TYPE E_CircuitBreakerStatus :
(
    READY := 0,         // Hazır
    OPERATING := 1,     // Hareket halinde
    INTERLOCKED := 2,   // Interlock aktif
    FAULTED := 3,       // Arızalı
    TRIPPED := 4,       // Trip durumunda
    NO_CONTROL := 5,    // PLC kontrol yok
    MAINTENANCE := 6    // Bakım gerekli
);
END_TYPE

(* stored: Version 1.1.0.1, ProductVersion 3.1.4024.15
   EnumerationTextList E_CircuitBreakerStatus: Id {8b66f4bb-02cd-4354-9c55-d481eb5f8d38} *)
